# B&R Automation Studio project WakeUpLight
Automation Studio 4.2.7.54 SP

## Configuration Config1

CPU X20CP1381, AutomationRuntime L4.10, Build 4.1.2, Vc V4.26.2

### Task classes (Cpu.sw)
```
Cyclic#4 (cycle 100000 us, tolerance 100000 us):
  light <- light.prg
Libraries: standard, AsArLog, runtime
```

### Hardware
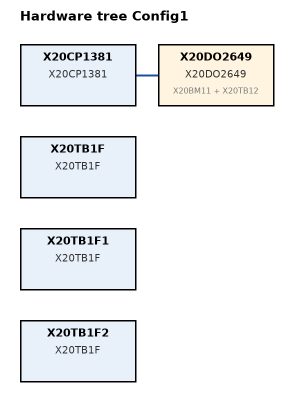
```
X20BM11 : X20BM11 v1.0.0.1  [X2X1 -> X20CP1381.IF6]
X20CP1381 : X20CP1381 v1.3.2.0  [X1 -> X1.SL; X2 -> X2.SL; X3 -> X3.SL]
  Module X1 (Type=X1, Virtual=true, Version=1.0.0.0)
    Connection (Connector=SS1, TargetModule=X20TB1F, TargetConnector=SS)
    Connection (Connector=SL, TargetModule=X20CP1381, TargetConnector=X1)
  Module X2 (Type=X2, Virtual=true, Version=1.0.0.0)
    Connection (Connector=SS1, TargetModule=X20TB1F1, TargetConnector=SS)
    Connection (Connector=SL, TargetModule=X20CP1381, TargetConnector=X2)
  Module X3 (Type=X3, Virtual=true, Version=1.0.0.0)
    Connection (Connector=SS1, TargetModule=X20TB1F2, TargetConnector=SS)
    Connection (Connector=SL, TargetModule=X20CP1381, TargetConnector=X3)
  Connector IF2:
    ActivateDevice = 1
    Mode = Manual
    InternetAddress = 192.168.0.10
    SubnetMask = 255.255.255.0
  ConfigurationID = svetlo_Config1
  TimerDeviceType = SWIOTIMER
  Cyclic1Duration = 10000
  Cyclic1Tolerance = 10000
  Cyclic2Duration = 20000
  Cyclic2Tolerance = 20000
  Cyclic3Duration = 50000
  Cyclic3Tolerance = 50000
  Cyclic4Duration = 100000
  Cyclic4Tolerance = 100000
  Cyclic5Duration = 200000
  Cyclic5Tolerance = 200000
  Cyclic6Duration = 500000
  Cyclic6Tolerance = 500000
  Cyclic7Duration = 1000000
  Cyclic7Tolerance = 1000000
  Cyclic8Duration = 10000
  Cyclic8Tolerance = 30000000
X20DO2649 : X20DO2649 v1.0.2.0  [SS1 -> X20TB12.SS; SL -> X20BM11.SL1]
X20TB12 : X20TB12 v1.0.0.0
X20TB1F : X20TB1F v1.0.0.0
X20TB1F1 : X20TB1F v1.0.0.0
X20TB1F2 : X20TB1F v1.0.0.0
```

### IoMap.iom - X20CP1381/IoMap.iom
```iecst
VAR_CONFIG
	::light:light AT %QX."X20DO2649".DigitalOutput02;
	::light:button AT %IX."X2".DigitalInput09;
END_VAR
```

## Logical view

Binary libraries used (declarations not repeated): operator, runtime, astime, AsIecCon, standard, AsArLog


### Program Logical/light (IEC)

#### Types.typ
```iecst
TYPE
	StateLight :
		(
		stateOutsideNightHours,
		stateOutOfBed,
		stateSleeping,
		stateFallingAsleep
		);
END_TYPE
```

#### Variables.var
```iecst
VAR
	light : BOOL;
	stateLight : StateLight;
	TON_0 : TON;
	button : BOOL;
	oldButton : BOOL;
	AsArLogWrite_0 : AsArLogWrite;
	oldStateLight : StateLight;
	stateEntered : BOOL;
	buttonPressed : BOOL;
	TP_0 : TP;
	speedFactor : INT;
	test : BOOL;
	DTStructureGetTime_0 : DTStructureGetTime;
	DTStructure1 : DTStructure;
	nightHours : BOOL;
END_VAR
```

#### Cyclic.st
```iecst
PROGRAM _CYCLIC

	IF test THEN
		speedFactor := 60;
	ELSE
		speedFactor := 1;
	END_IF

	TP_0(IN := button <> oldButton, PT := T#500ms);
	buttonPressed := EDGEPOS(TP_0.Q);
	oldButton := button;

	DTStructureGetTime_0(enable := 1, pDTStructure := ADR(DTStructure1));

	IF DTStructure1.hour >= 6 AND DTStructure1.hour < 20 THEN
		nightHours := FALSE;
	ELSE
		nightHours := TRUE;
	END_IF

	IF test THEN
		nightHours := TRUE;
	END_IF

	IF NOT nightHours THEN
		stateLight := stateOutsideNightHours;
	END_IF

	CASE stateLight OF

		stateOutsideNightHours:

			IF stateEntered THEN
				AsArLogWrite_0.enable := TRUE;
				AsArLogWrite_0.asciiString := ADR('outside night hours');
			END_IF

			IF nightHours THEN
				stateLight := stateOutOfBed;
			END_IF

			light := FALSE;

		stateOutOfBed:

			IF stateEntered THEN
				AsArLogWrite_0.enable := TRUE;
				AsArLogWrite_0.asciiString := ADR('out of bed');
			END_IF

			TON_0(IN := TRUE, PT := T#1s);
			IF TON_0.Q THEN
				light := TRUE;
			ELSE
				light := FALSE;
			END_IF

			IF buttonPressed THEN
				stateLight := stateFallingAsleep;
			END_IF

		stateSleeping:

			IF stateEntered THEN
				AsArLogWrite_0.enable := TRUE;
				AsArLogWrite_0.asciiString := ADR('sleeping');
				light := TRUE;
			END_IF

			IF light THEN
				TON_0(IN := TRUE, PT := T#5m/speedFactor);
				IF TON_0.Q THEN
					TON_0(IN := FALSE);
					light := FALSE;
				END_IF
			ELSE
				TON_0(IN := TRUE, PT := T#15m/speedFactor);
				IF TON_0.Q THEN
					TON_0(IN := FALSE);
					light := TRUE;
				END_IF
			END_IF

			IF buttonPressed THEN
				stateLight := stateOutOfBed;
			END_IF

		stateFallingAsleep:

			IF stateEntered THEN
				AsArLogWrite_0.enable := TRUE;
				AsArLogWrite_0.asciiString := ADR('falling asleep');
			END_IF

			TON_0(IN := TRUE, PT := T#20m/speedFactor);

			IF TON_0.Q THEN
				stateLight := stateSleeping;
			END_IF

			IF buttonPressed THEN
				stateLight := stateOutOfBed;
			END_IF

			light := FALSE;

	END_CASE

	IF oldStateLight <> stateLight THEN
		TON_0(IN := FALSE);
		stateEntered := TRUE;
	ELSE
		stateEntered := FALSE;
	END_IF

	AsArLogWrite_0(ident := arlogBASE_USER_LOG_IDENT, mem:=ADR(stateLight), len:= SIZEOF(oldStateLight), logLevel := arlogLEVEL_INFO);
	IF AsArLogWrite_0.status = 0 THEN
		AsArLogWrite_0.enable := FALSE;
	END_IF

	oldStateLight := stateLight;

END_PROGRAM
```

Listed in the project but not available here: Logical/Global.typ, Logical/Global.var
